// TIA Portal V19 export
DATA_BLOCK "LB212_FeedA02"   // DB148
// stored: InstanceOfName ButtonsSafe_LB212_FeedA02, InstanceOfType FB
"ButtonsSafe_LB212_FeedA02"
   // VAR_INPUT
   //    Reset_OthersPBs_Activation_IN : Bool;
   // END_VAR
   // VAR_OUTPUT
   //    Reset_OthersPBs_Activation_OUT : Bool;
   // END_VAR
   // VAR
   //    i : Int;
   //    iOperation : Int;
   //    iConcurrentOperation : Int;
   //    SettingWriteDone : Bool;
   //    PbPanel : "Buttons2Hands";
   //    PB : Struct
   //       ResetAlarms : Bool;
   //       Rollformer_Bwd : Bool;
   //       Rollformer_Fwd : Bool;
   //    END_STRUCT;
   // END_VAR
BEGIN
END_DATA_BLOCK
